PROGRAM MAIN
VAR
END_VAR

SEQ.iStepN:=25;
POU();
Water_Tank();
POU_1();
POU_3();
SequencyControl();
ValveControl();

END_PROGRAM

(* stored: Version 1.1.0.1, ProductVersion 3.1.4024.12
   POU MAIN: Id {2c837950-4eeb-403d-b549-a1fa9ff09b39}, SpecialFunc None *)
